PROGRAM Axis04_Set_Work_End_Speed
VAR
END_VAR


IF GVL_System.Manual_Mode THEN 
	GVL_Axis04.Work_End_Speed := 30 ;
ELSE 
	GVL_Axis04.Work_End_Speed:= 60;
END_IF

END_PROGRAM

(* stored: Version 1.1.0.1, ProductVersion 3.1.4024.16
   POU Axis04_Set_Work_End_Speed: Id {e32a4f33-ffb8-4eef-8cba-292e6d0e32cd}, SpecialFunc None *)
